INTERFACE ITF_Schuif_DigOutOpen_AFO

METHOD set : BOOL
VAR_INPUT
END_VAR
END_METHOD

END_INTERFACE

(* stored: Version 1.1.0.1, ProductVersion 3.1.4026.8
   Itf ITF_Schuif_DigOutOpen_AFO: Id {54c54e13-a755-4a5f-809c-de1feb8e1e8a}
   Method set: Id {3e24cccd-bdea-48e9-8ad2-444d2cb582b4} *)
